Universal Robots URScript: 00B_03_Che_ZhuaXian.script

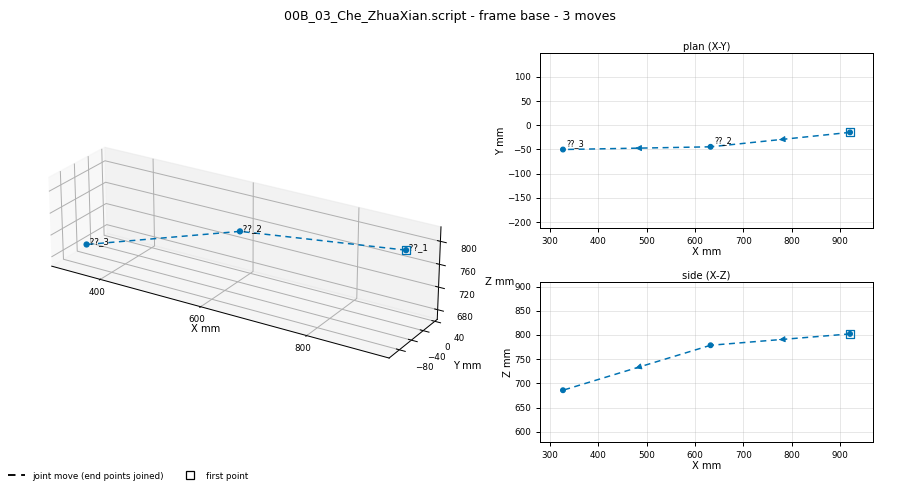
[picture p0: tool path of 00B_03_Che_ZhuaXian.script in frame base, 3 of 3 moves have a stored position in this frame; points joined in program order, loops and branches not executed]
def P00B_03_Che_ZhuaXian():
  set_gravity([0.0, 0.0, 9.82])
  set_safety_mode_transition_hardness(1)
  set_standard_analog_input_domain(0, 1)
  set_standard_analog_input_domain(1, 1)
  set_tool_analog_input_domain(0, 1)
  set_tool_analog_input_domain(1, 1)
  set_analog_outputdomain(0, 0)
  set_analog_outputdomain(1, 0)
  set_tool_voltage(24)
  set_input_actions_to_default()
  set_tcp(p[0.0,0.0,0.32,0.0,0.0,-0.5236])
  set_payload(8.0)
  global Zhua_1=[0.08063, -2.42649, -1.72682, -0.47876, 0.40808, -1.10831]
  global prepose=p[0.98979, -0.16931, -0.39963, 1.98720, 0.07234, 0.05469]
  global i_var_2=0
  global i_var_1=True
  global pose=p[0.98979, -0.31931, -0.39963, 1.98720, 0.07234, 0.05469]
  $ 1 "机器人程序"
  $ 2 "MoveJ"
  $ 3 "路点_1"
  set_tcp(p[0.0,0.0,0.32,0.0,0.0,-0.5236])
  movej(get_inverse_kin(p[.920325694299, -.014751913315, .802090726890, 1.103725960549, 1.210647533545, 1.370058891584], qnear=[0.1848503053188324, -1.4502208868609827, -1.439040486012594, -3.297612015401022, -1.5013678709613245, 0.5357873439788818]), a=0.6981317007977318, v=0.5235987755982988)
  $ 4 "路点_2"
  set_tcp(p[0.0,0.0,0.32,0.0,0.0,-0.5236])
  movej(get_inverse_kin(p[.632242339591, -.044597837813, .778614894906, 1.103717556783, 1.210551154493, 1.369917607725], qnear=[0.306870698928833, -0.9581745306598108, -1.777787987385885, -3.4486516157733362, -1.3784735838519495, 0.5276882648468018]), a=0.6981317007977318, v=0.5235987755982988)
  $ 5 "路点_3"
  set_tcp(p[0.0,0.0,0.32,0.0,0.0,-0.5236])
  movej(get_inverse_kin(p[.327313234849, -.050214348130, .685717824622, -.037506490724, .082952000942, 1.218561413578], qnear=[0.2739230692386627, -1.172699276600973, -2.7697015444384974, -0.8335326353656214, -1.6334694067584437, -0.1052473227130335]), a=0.6981317007977318, v=0.5235987755982988)
end
